PROGRAM MAIN
VAR
END_VAR

END_PROGRAM

(* stored: Version 1.1.0.1
   POU MAIN: Id {963367b4-7853-46d9-a119-421c43f5684c} *)
